FUNCTION_BLOCK Calamity (* CAT Function Block Type *)
  (* Standard: 61499-2 *)
  (* Version 0.0, 6/21/2026, Schneider Electric, template *)
  PACKAGE SE.Nereda;
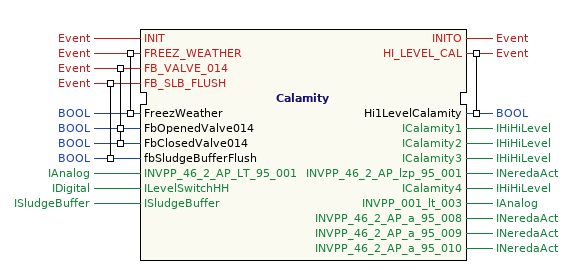
  EVENT_INPUT
    INIT;
    FREEZ_WEATHER WITH FreezWeather;
    FB_VALVE_014 WITH FbOpenedValve014, FbClosedValve014;
    FB_SLB_FLUSH WITH fbSludgeBufferFlush;
  END_EVENT
  EVENT_OUTPUT
    INITO;
    HI_LEVEL_CAL WITH Hi1LevelCalamity; (* Input changed *)
  END_EVENT
  VAR_INPUT
    FreezWeather : BOOL;
    FbOpenedValve014 : BOOL;
    FbClosedValve014 : BOOL;
    fbSludgeBufferFlush : BOOL;
  END_VAR
  VAR_OUTPUT
    Hi1LevelCalamity : BOOL; (* Output value *)
  END_VAR
  SOCKETS
    INVPP_46_2_AP_LT_95_001 : IAnalog;
    ILevelSwitchHH : IDigital;
    ISludgeBuffer : ISludgeBuffer;
  END_SOCKETS
  PLUGS
    ICalamity1 : IHiHiLevel;
    ICalamity2 : IHiHiLevel;
    ICalamity3 : IHiHiLevel;
    INVPP_46_2_AP_lzp_95_001 : INeredaAct;
    ICalamity4 : IHiHiLevel;
    INVPP_001_lt_003 : IAnalog;
  END_PLUGS
  PLUGS
    INVPP_46_2_AP_a_95_008 : INeredaAct;
    INVPP_46_2_AP_a_95_009 : INeredaAct;
    INVPP_46_2_AP_a_95_010 : INeredaAct;
  END_PLUGS
  (* 01 - FUNCTIONNAL INPUT INTERFACE *)
  (* 00 - INITIALIZATION *)
  (* 05 - LOGIC *)
  (* 06 - HMI INTERFACE *)
  (* 03 - FIELD INTERFACE *)
  (* Calamity Pump Logic *)
  (* 02 - FUNCTIONNAL OUTPUT INTERFACE *)
  (* Calamity Valves Control *)
  FBS
    IThis : Calamity_HMI(QI := TRUE);
    CalamityPumpLogic : CalamityPumpBasic;
    NVPP_46_2_AP_LT_95_001_Status : decodeStatus; {SET_ATTRIBUTE(Configuration.Component.HideUnusedPorts, )}
    PumpCmd : boolValueChanged;
    CMD_NVPP_46_2_AP_a_95_008 : CalamityValveLogic;
    CMD_NVPP_46_2_AP_a_95_009 : CalamityValveLogic;
    CMD_NVPP_46_2_AP_a_95_010 : CalamityValveLogic;
    H1Level : COMPARE_1329C2AB45109BAAB; {SET_ATTRIBUTE(Configuration.GenericFBType.InterfaceParams, Runtime.Standard#CNT:=2;IN${CNT$}:REAL)} {SET_ATTRIBUTE(Configuration.Component.HideUnusedPorts, )}
    HiLevelSmooth : boolValueChanged;
    CalamityPump : BOOL2INT;
    LevelSwitchHH : INT2BOOL;
  END_FBS
  EVENT_CONNECTIONS
    INVPP_46_2_AP_LT_95_001.REQ_STATUS TO NVPP_46_2_AP_LT_95_001_Status.REQ;
    INVPP_46_2_AP_LT_95_001.REQ TO H1Level.REQ;
    H1Level.CNF TO HiLevelSmooth.REQ;
    INIT TO IThis.AABF4BC3AB55D4F4;
    HiLevelSmooth.CHD TO IThis.A0CAD0828CA5CECC;
    INVPP_46_2_AP_LT_95_001.REQ TO IThis.04D261C42461D5AD;
    NVPP_46_2_AP_LT_95_001_Status.CNF TO IThis.84CA074A02EC9398;
    IThis.22CD6E75BAD411C6 TO H1Level.REQ;
    HiLevelSmooth.CHD TO HI_LEVEL_CAL;
    CMD_NVPP_46_2_AP_a_95_010.599C3061E75F42AF TO INITO;
    NVPP_46_2_AP_LT_95_001_Status.CNF TO ICalamity1.15126F43E529BB4F;
    NVPP_46_2_AP_LT_95_001_Status.CNF TO ICalamity2.15126F43E529BB4F;
    NVPP_46_2_AP_LT_95_001_Status.CNF TO ICalamity3.15126F43E529BB4F;
    NVPP_46_2_AP_LT_95_001_Status.CNF TO ICalamity4.15126F43E529BB4F;
    NVPP_46_2_AP_LT_95_001_Status.CNF TO CalamityPumpLogic.DF23DCB361DA9198;
    ILevelSwitchHH.REQ TO LevelSwitchHH.DD5870AA881150BB;
    LevelSwitchHH.6FC99A5BD1C38561 TO IThis.84CA074A02EC9398;
    LevelSwitchHH.6FC99A5BD1C38561 TO ICalamity1.15126F43E529BB4F;
    LevelSwitchHH.6FC99A5BD1C38561 TO ICalamity2.15126F43E529BB4F;
    LevelSwitchHH.6FC99A5BD1C38561 TO ICalamity3.15126F43E529BB4F;
    LevelSwitchHH.6FC99A5BD1C38561 TO ICalamity4.15126F43E529BB4F;
    FB_SLB_FLUSH TO ISludgeBuffer.6E1E38EF865F33B9;
    ISludgeBuffer.53832F2A5D6ADA0F TO CMD_NVPP_46_2_AP_a_95_008.D723ED8511816BBA;
    ISludgeBuffer.E7834F57A023D9E9 TO INVPP_001_lt_003.REQ;
    ISludgeBuffer.C4552068F0BCC726 TO INVPP_001_lt_003.REQ_STATUS;
    FREEZ_WEATHER TO CMD_NVPP_46_2_AP_a_95_009.69A24641938E98BB;
    FREEZ_WEATHER TO CMD_NVPP_46_2_AP_a_95_008.69A24641938E98BB;
    FREEZ_WEATHER TO CMD_NVPP_46_2_AP_a_95_010.69A24641938E98BB;
    FB_VALVE_014 TO CMD_NVPP_46_2_AP_a_95_009.D723ED8511816BBA;
    IThis.641BD1E2D34D3C2A TO CalamityPumpLogic.C88AF9BE306E1559;
    INVPP_46_2_AP_lzp_95_001.9CD053F8408797ED TO CalamityPumpLogic.6E6C941905C3D56D;
    INVPP_46_2_AP_lzp_95_001.CC753684FA882790 TO CalamityPumpLogic.6E6C941905C3D56D;
    CalamityPumpLogic.D80113876A820D78 TO PumpCmd.REQ;
    CalamityPumpLogic.D0E3147DF23F35C3 TO INVPP_46_2_AP_lzp_95_001.1E00729184986247;
    CalamityPumpLogic.65B8E9E9FD40924C TO IThis.5C91736D821E7D87;
    PumpCmd.CHD TO CalamityPump.DD5870AA881150BB;
    CalamityPump.6FC99A5BD1C38561 TO INVPP_46_2_AP_lzp_95_001.0F1CDF9A9B4A227A;
    IThis.67A10949F5B1AAAB TO CMD_NVPP_46_2_AP_a_95_008.B0D405FAB24B1E1C;
    CMD_NVPP_46_2_AP_a_95_008.599C3061E75F42AF TO CMD_NVPP_46_2_AP_a_95_009.B0D405FAB24B1E1C;
    CMD_NVPP_46_2_AP_a_95_009.599C3061E75F42AF TO CMD_NVPP_46_2_AP_a_95_010.B0D405FAB24B1E1C;
    CMD_NVPP_46_2_AP_a_95_010.599C3061E75F42AF TO IThis.5F30A434EE074757;
    INVPP_46_2_AP_lzp_95_001.9CD053F8408797ED TO CMD_NVPP_46_2_AP_a_95_010.D723ED8511816BBA;
  END_CONNECTIONS
  DATA_CONNECTIONS
    INVPP_46_2_AP_LT_95_001.Status TO NVPP_46_2_AP_LT_95_001_Status.Status;
    INVPP_46_2_AP_LT_95_001.Value TO H1Level.IN1;
    H1Level.GE TO HiLevelSmooth.Input;
    HiLevelSmooth.Output TO IThis.A0529EAA411F2CC1;
    INVPP_46_2_AP_LT_95_001.Value TO IThis.CC24354046456B52;
    INVPP_46_2_AP_LT_95_001.ValueMin TO IThis.6CD4081C3EBA3A32;
    INVPP_46_2_AP_LT_95_001.ValueMax TO IThis.9EA72B9C2F54520D;
    NVPP_46_2_AP_LT_95_001_Status.HiHiAlarm TO IThis.DB178D55CCC36649;
    IThis.AEE53212905D5ECF TO H1Level.IN2;
    HiLevelSmooth.Output TO Hi1LevelCalamity;
    NVPP_46_2_AP_LT_95_001_Status.HiHiAlarm TO ICalamity1.C818324478A2F205;
    NVPP_46_2_AP_LT_95_001_Status.HiHiAlarm TO ICalamity2.C818324478A2F205;
    NVPP_46_2_AP_LT_95_001_Status.HiHiAlarm TO ICalamity3.C818324478A2F205;
    NVPP_46_2_AP_LT_95_001_Status.HiHiAlarm TO ICalamity4.C818324478A2F205;
    NVPP_46_2_AP_LT_95_001_Status.HiAlarm TO CalamityPumpLogic.F3BCD1558E816D4D;
    NVPP_46_2_AP_LT_95_001_Status.LoAlarm TO CalamityPumpLogic.5E4B50A6B54508F9;
    ILevelSwitchHH.Value TO LevelSwitchHH.4573FC8F228EB71D;
    LevelSwitchHH.A6DEF5F9C27C1848 TO IThis.2EF3EC59F5FC7236;
    LevelSwitchHH.A6DEF5F9C27C1848 TO ICalamity1.96B50ADF37756FFC;
    LevelSwitchHH.A6DEF5F9C27C1848 TO ICalamity2.96B50ADF37756FFC;
    LevelSwitchHH.A6DEF5F9C27C1848 TO ICalamity3.96B50ADF37756FFC;
    LevelSwitchHH.A6DEF5F9C27C1848 TO ICalamity4.96B50ADF37756FFC;
    fbSludgeBufferFlush TO ISludgeBuffer.42FB791008946C6C;
    ISludgeBuffer.AEFD07E0C2212479 TO CMD_NVPP_46_2_AP_a_95_008.859CB6DCE329D25D;
    ISludgeBuffer.7C3414AE091CC670 TO CMD_NVPP_46_2_AP_a_95_008.985B4AC3F5EAC315;
    ISludgeBuffer.98ED49B8E6019185 TO INVPP_001_lt_003.Value;
    ISludgeBuffer.C5E968D74BD846AF TO INVPP_001_lt_003.ValueMin;
    ISludgeBuffer.C09AFDABE4AE7C73 TO INVPP_001_lt_003.ValueMax;
    ISludgeBuffer.3AE62655EE14D04A TO INVPP_001_lt_003.Status;
    FreezWeather TO CMD_NVPP_46_2_AP_a_95_009.CF9FAF2BC0E65782;
    FreezWeather TO CMD_NVPP_46_2_AP_a_95_008.CF9FAF2BC0E65782;
    FreezWeather TO CMD_NVPP_46_2_AP_a_95_010.CF9FAF2BC0E65782;
    FbOpenedValve014 TO CMD_NVPP_46_2_AP_a_95_009.859CB6DCE329D25D;
    FbClosedValve014 TO CMD_NVPP_46_2_AP_a_95_009.985B4AC3F5EAC315;
    IThis.DD5B1A7D95503A0A TO CalamityPumpLogic.4B740182EAB3F037;
    INVPP_46_2_AP_lzp_95_001.B762734C094A7162 TO CalamityPumpLogic.FFFB2DFE6F24B566;
    INVPP_46_2_AP_lzp_95_001.D83B5BDEFA4D797C TO CalamityPumpLogic.19DC18FF464DA580;
    INVPP_46_2_AP_lzp_95_001.8A8A07EFCDA1443C TO CalamityPumpLogic.126DEC6100818E4D;
    CalamityPumpLogic.26811D54DFA4688D TO PumpCmd.Input;
    CalamityPumpLogic.A806F58E43A04127 TO INVPP_46_2_AP_lzp_95_001.1BC103921BBFDA0B;
    CalamityPumpLogic.E48FF2B0215DCB21 TO IThis.8E6BDAE3BC6A4EA4;
    PumpCmd.Output TO CalamityPump.4573FC8F228EB71D;
    CalamityPump.A6DEF5F9C27C1848 TO INVPP_46_2_AP_lzp_95_001.710D7FC54EE3F35A;
    INVPP_46_2_AP_lzp_95_001.D83B5BDEFA4D797C TO CMD_NVPP_46_2_AP_a_95_010.985B4AC3F5EAC315;
    INVPP_46_2_AP_lzp_95_001.B762734C094A7162 TO CMD_NVPP_46_2_AP_a_95_010.859CB6DCE329D25D;
  END_CONNECTIONS
  ADAPTER_CONNECTIONS
    CMD_NVPP_46_2_AP_a_95_008.F83096AD3BF61126 TO INVPP_46_2_AP_a_95_008;
    CMD_NVPP_46_2_AP_a_95_009.F83096AD3BF61126 TO INVPP_46_2_AP_a_95_009;
    CMD_NVPP_46_2_AP_a_95_010.F83096AD3BF61126 TO INVPP_46_2_AP_a_95_010;
  END_CONNECTIONS
END_FUNCTION_BLOCK
